// TIA Portal V20 export
DATA_BLOCK "BK03"   // DB316
// stored: MemoryReserve 100
   VAR
      "X10-1.SUCTION PAD TOP LEFT PRESSURE SWITCH" : Bool := FALSE;
      "X10-2.SUCTION PAD TOP RIGHT PRESSURE SWITCH" : Bool := FALSE;
      "X12-1.SUCTION PAD BTM LEFT PRESSURE SWITCH" : Bool := FALSE;
      "X12-2.SUCTION PAD BTM RIGHT PRESSURE SWITCH" : Bool := FALSE;
      "X14-1.SUCTION PAD TOP TAPE PRESSURE SWITCH" : Bool := FALSE;
      "X14-2.SUCTION PAD BTM TAPE PRESSURE SWITCH" : Bool := FALSE;
      "X16-1.ROTATION SAFETY PIN POSITION" : Bool := TRUE;
      "X16-2.SPARE" : Bool := FALSE;
   END_VAR
BEGIN
END_DATA_BLOCK
